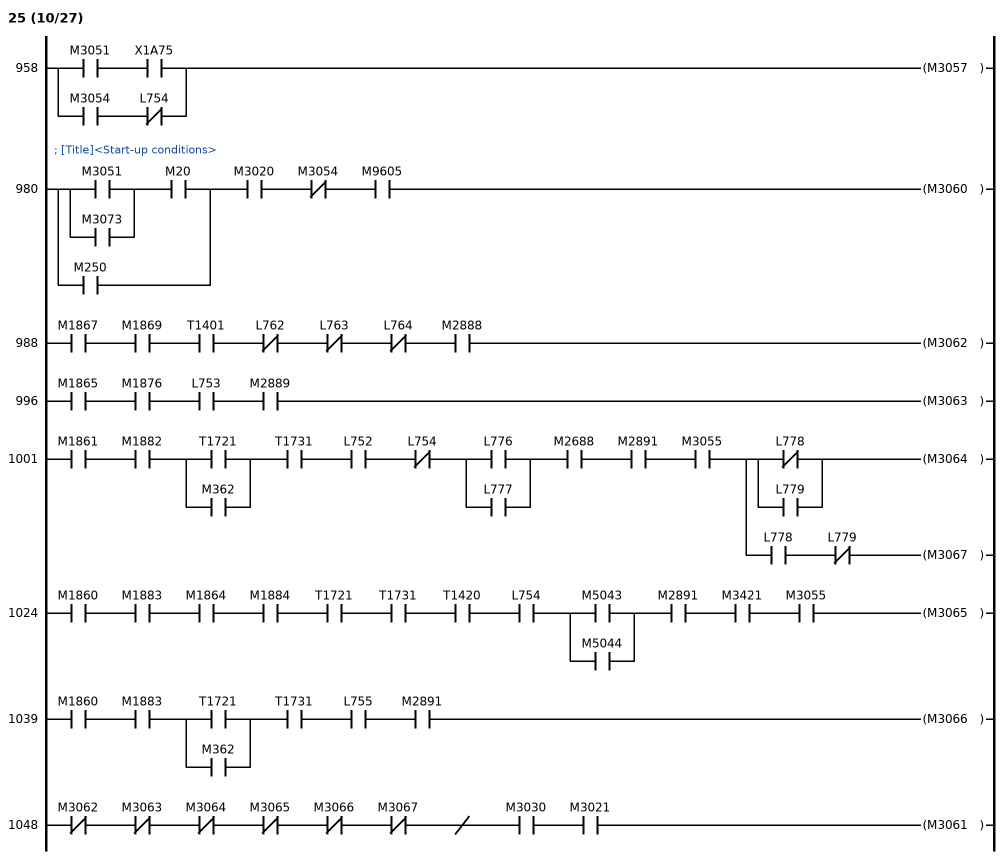
958   LD      M3051
      AND     X1A75
      LD      M3054
      ANI     L754
      ORB
      OUT     M3057
; [Title]<Start-up conditions>
980   LD      M3051
      OR      M3073
      AND     M20
      OR      M250
      AND     M3020
      ANI     M3054
      AND     M9605
      OUT     M3060
988   LD      M1867
      AND     M1869
      AND     T1401
      ANI     L762
      ANI     L763
      ANI     L764
      AND     M2888
      OUT     M3062
996   LD      M1865
      AND     M1876
      AND     L753
      AND     M2889
      OUT     M3063
1001  LD      M1861
      AND     M1882
      LD      T1721
      OR      M362
      ANB
      AND     T1731
      AND     L752
      ANI     L754
      LD      L776
      OR      L777
      ANB
      AND     M2688
      AND     M2891
      AND     M3055
      MPS
      LDI     L778
      OR      L779
      ANB
      OUT     M3064
      MPP
      AND     L778
      ANI     L779
      OUT     M3067
1024  LD      M1860
      AND     M1883
      AND     M1864
      AND     M1884
      AND     T1721
      AND     T1731
      AND     T1420
      AND     L754
      LD      M5043
      OR      M5044
      ANB
      AND     M2891
      AND     M3421
      AND     M3055
      OUT     M3065
1039  LD      M1860
      AND     M1883
      LD      T1721
      OR      M362
      ANB
      AND     T1731
      AND     L755
      AND     M2891
      OUT     M3066
1048  LDI     M3062
      ANI     M3063
      ANI     M3064
      ANI     M3065
      ANI     M3066
      ANI     M3067
      INV
      AND     M3030
      AND     M3021
      OUT     M3061
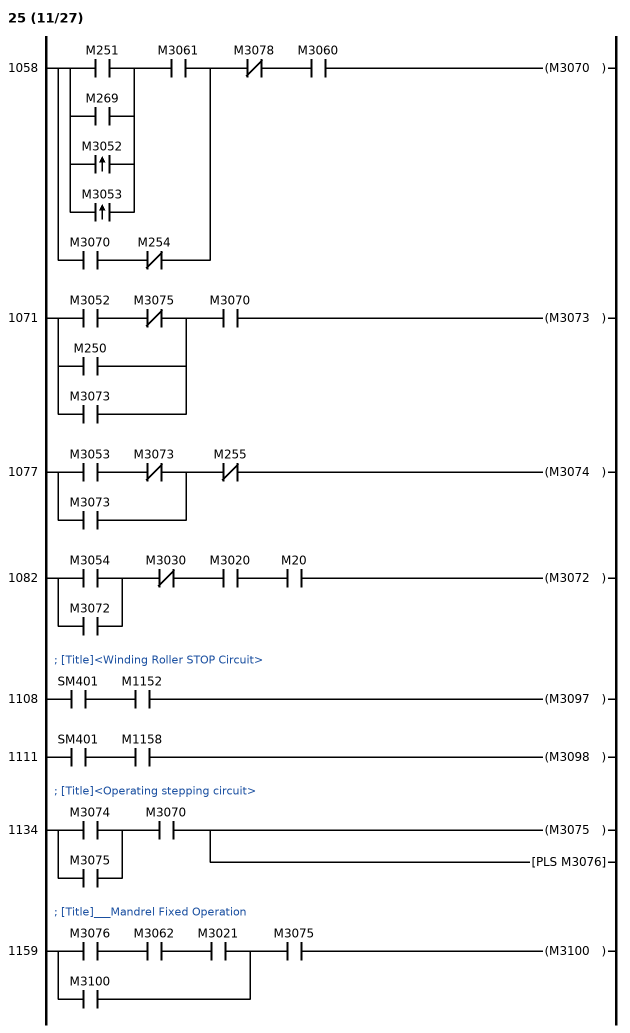
1058  LD      M251
      OR      M269
      ORP     M3052
      ORP     M3053
      AND     M3061
      LD      M3070
      ANI     M254
      ORB
      ANI     M3078
      AND     M3060
      OUT     M3070
1071  LD      M3052
      ANI     M3075
      OR      M250
      OR      M3073
      AND     M3070
      OUT     M3073
1077  LD      M3053
      ANI     M3073
      OR      M3073
      ANI     M255
      OUT     M3074
1082  LD      M3054
      OR      M3072
      ANI     M3030
      AND     M3020
      AND     M20
      OUT     M3072
; [Title]<Winding Roller STOP Circuit>
1108  LD      SM401
      AND     M1152
      OUT     M3097
1111  LD      SM401
      AND     M1158
      OUT     M3098
; [Title]<Operating stepping circuit>
1134  LD      M3074
      OR      M3075
      AND     M3070
      OUT     M3075
      PLS     M3076
; [Title]___Mandrel Fixed Operation
1159  LD      M3076
      AND     M3062
      AND     M3021
      OR      M3100
      AND     M3075
      OUT     M3100
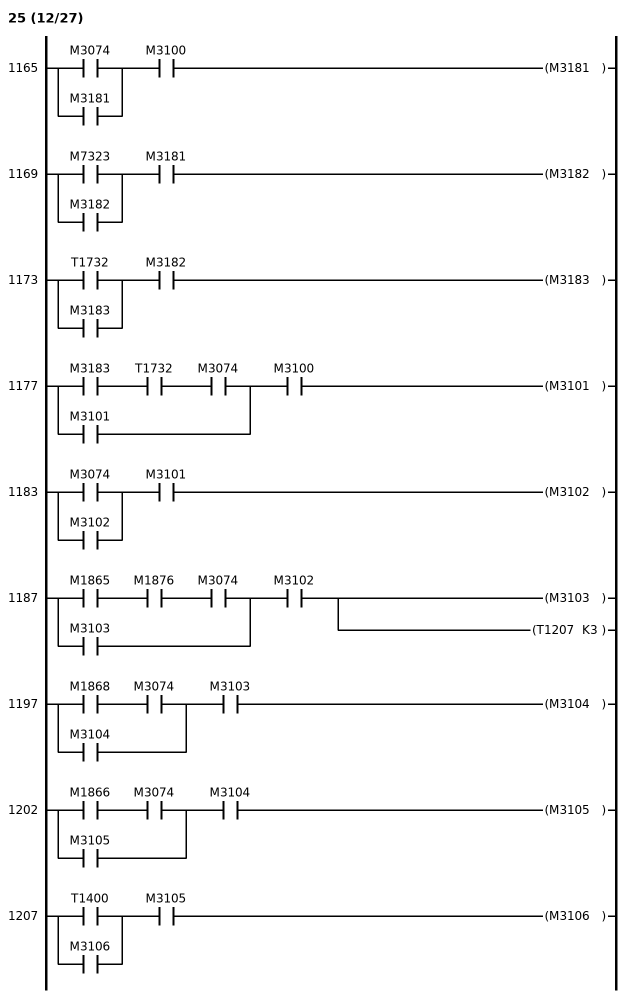
1165  LD      M3074
      OR      M3181
      AND     M3100
      OUT     M3181
1169  LD      M7323
      OR      M3182
      AND     M3181
      OUT     M3182
1173  LD      T1732
      OR      M3183
      AND     M3182
      OUT     M3183
1177  LD      M3183
      AND     T1732
      AND     M3074
      OR      M3101
      AND     M3100
      OUT     M3101
1183  LD      M3074
      OR      M3102
      AND     M3101
      OUT     M3102
1187  LD      M1865
      AND     M1876
      AND     M3074
      OR      M3103
      AND     M3102
      OUT     M3103
      OUT     T1207 K3
1197  LD      M1868
      AND     M3074
      OR      M3104
      AND     M3103
      OUT     M3104
1202  LD      M1866
      AND     M3074
      OR      M3105
      AND     M3104
      OUT     M3105
1207  LD      T1400
      OR      M3106
      AND     M3105
      OUT     M3106
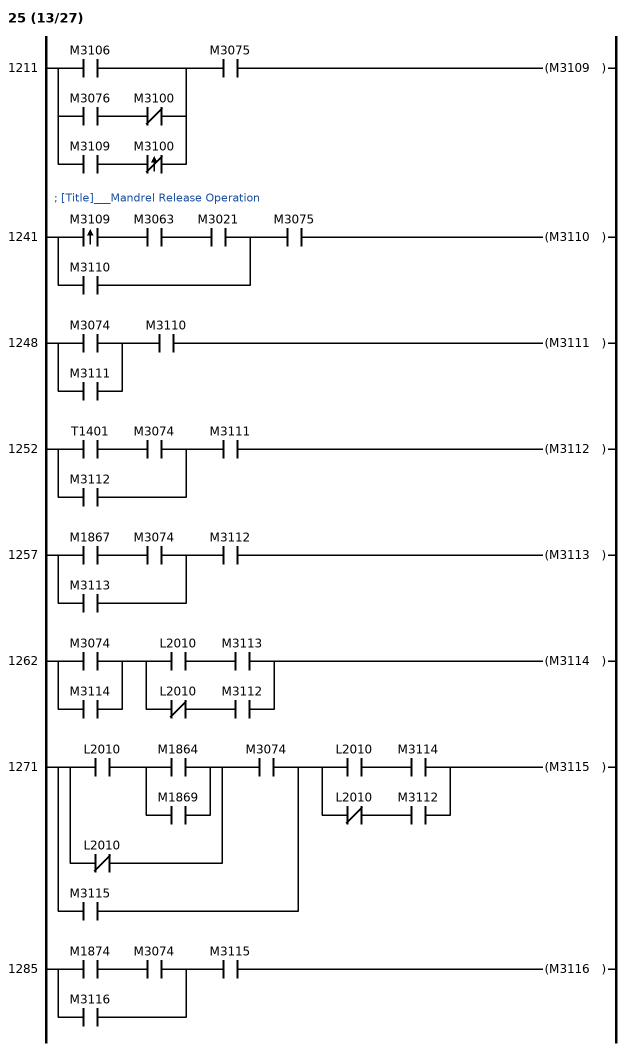
1211  LD      M3106
      LD      M3076
      ANI     M3100
      ORB
      LD      M3109
      ANDPI   M3100
      ORB
      AND     M3075
      OUT     M3109
; [Title]___Mandrel Release Operation
1241  LDP     M3109
      AND     M3063
      AND     M3021
      OR      M3110
      AND     M3075
      OUT     M3110
1248  LD      M3074
      OR      M3111
      AND     M3110
      OUT     M3111
1252  LD      T1401
      AND     M3074
      OR      M3112
      AND     M3111
      OUT     M3112
1257  LD      M1867
      AND     M3074
      OR      M3113
      AND     M3112
      OUT     M3113
1262  LD      M3074
      OR      M3114
      LD      L2010
      AND     M3113
      LDI     L2010
      AND     M3112
      ORB
      ANB
      OUT     M3114
1271  LD      L2010
      LD      M1864
      OR      M1869
      ANB
      ORI     L2010
      AND     M3074
      OR      M3115
      LD      L2010
      AND     M3114
      LDI     L2010
      AND     M3112
      ORB
      ANB
      OUT     M3115
1285  LD      M1874
      AND     M3074
      OR      M3116
      AND     M3115
      OUT     M3116
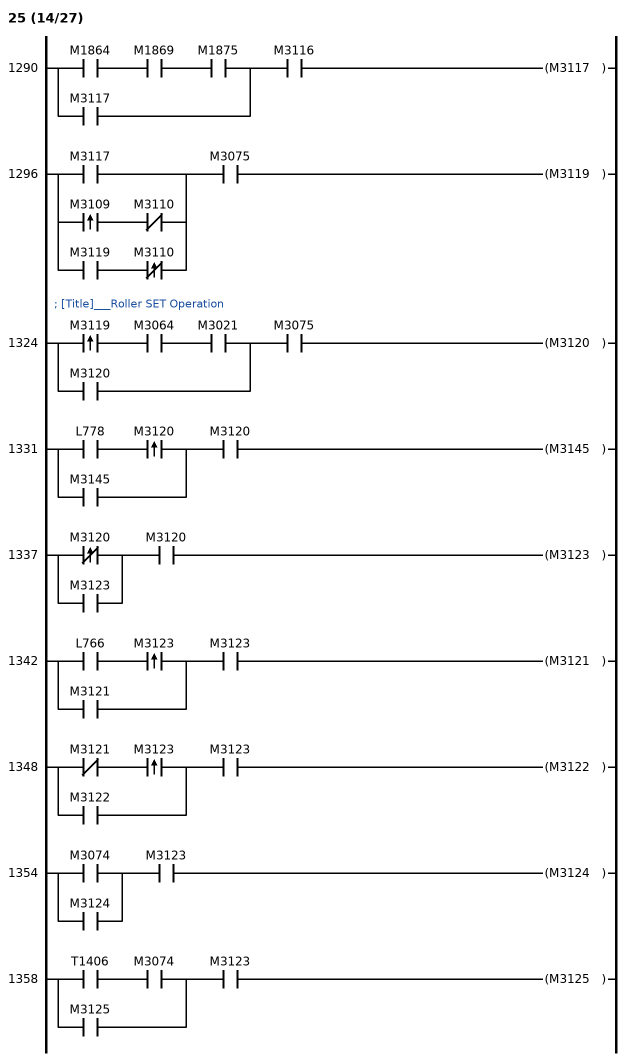
1290  LD      M1864
      AND     M1869
      AND     M1875
      OR      M3117
      AND     M3116
      OUT     M3117
1296  LD      M3117
      LDP     M3109
      ANI     M3110
      ORB
      LD      M3119
      ANDPI   M3110
      ORB
      AND     M3075
      OUT     M3119
; [Title]___Roller SET Operation
1324  LDP     M3119
      AND     M3064
      AND     M3021
      OR      M3120
      AND     M3075
      OUT     M3120
1331  LD      L778
      ANDP    M3120
      OR      M3145
      AND     M3120
      OUT     M3145
1337  LDPI    M3120
      OR      M3123
      AND     M3120
      OUT     M3123
1342  LD      L766
      ANDP    M3123
      OR      M3121
      AND     M3123
      OUT     M3121
1348  LDI     M3121
      ANDP    M3123
      OR      M3122
      AND     M3123
      OUT     M3122
1354  LD      M3074
      OR      M3124
      AND     M3123
      OUT     M3124
1358  LD      T1406
      AND     M3074
      OR      M3125
      AND     M3123
      OUT     M3125
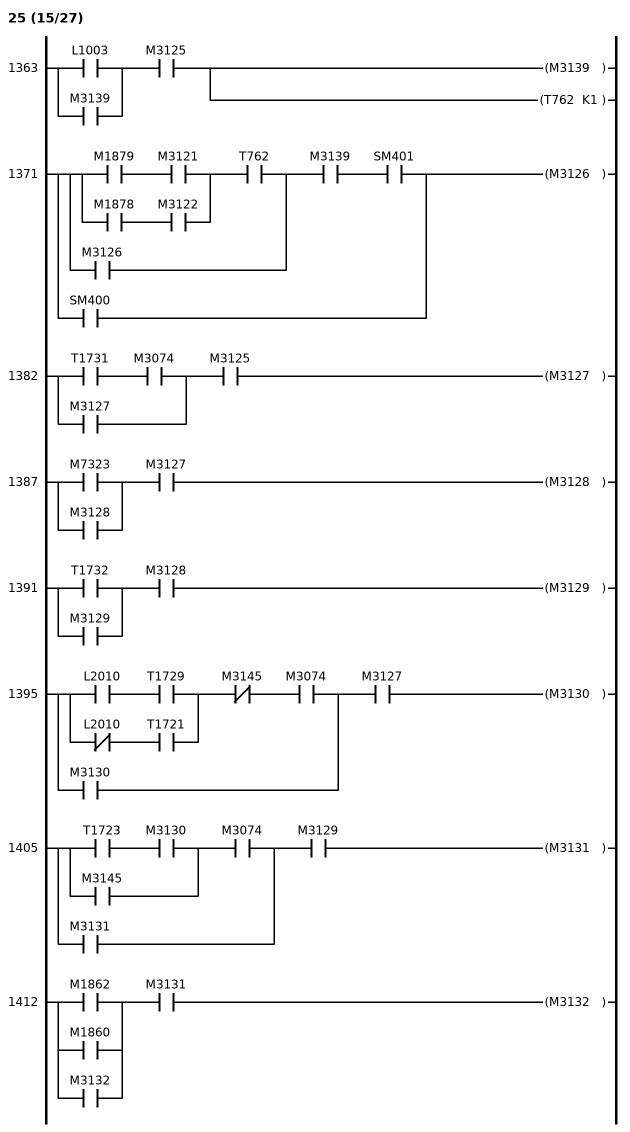
1363  LD      L1003
      OR      M3139
      AND     M3125
      OUT     M3139
      OUT     T762 K1
1371  LD      M1879
      AND     M3121
      LD      M1878
      AND     M3122
      ORB
      AND     T762
      OR      M3126
      AND     M3139
      AND     SM401
      OR      SM400
      OUT     M3126
1382  LD      T1731
      AND     M3074
      OR      M3127
      AND     M3125
      OUT     M3127
1387  LD      M7323
      OR      M3128
      AND     M3127
      OUT     M3128
1391  LD      T1732
      OR      M3129
      AND     M3128
      OUT     M3129
1395  LD      L2010
      AND     T1729
      LDI     L2010
      AND     T1721
      ORB
      ANI     M3145
      AND     M3074
      OR      M3130
      AND     M3127
      OUT     M3130
1405  LD      T1723
      AND     M3130
      OR      M3145
      AND     M3074
      OR      M3131
      AND     M3129
      OUT     M3131
1412  LD      M1862
      OR      M1860
      OR      M3132
      AND     M3131
      OUT     M3132
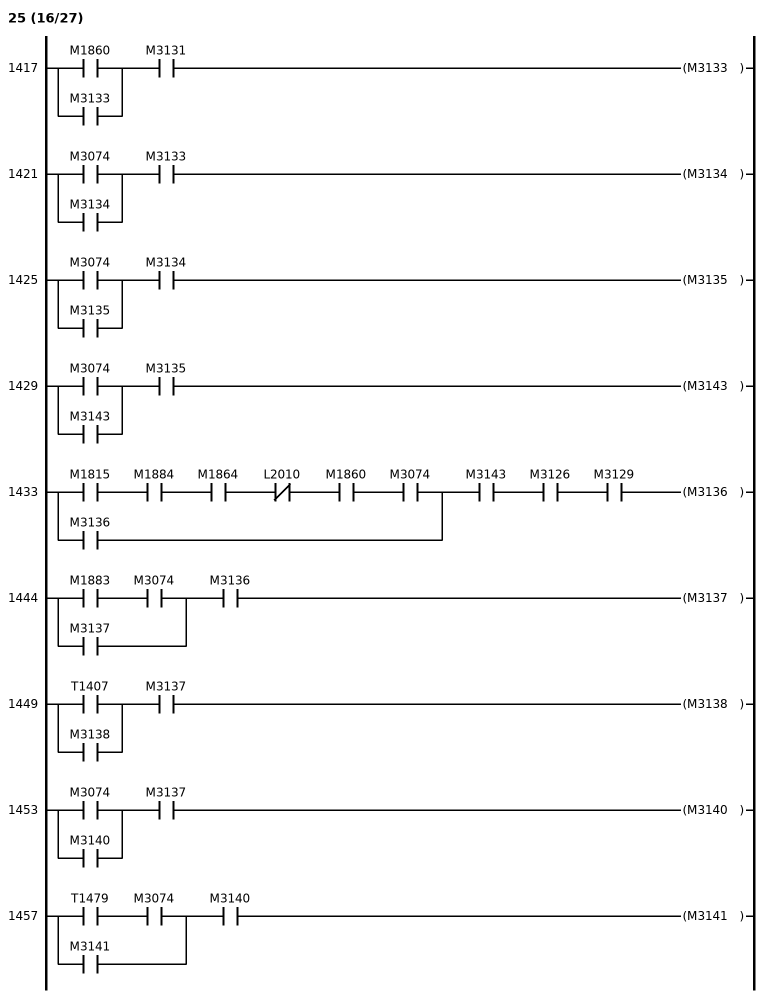
1417  LD      M1860
      OR      M3133
      AND     M3131
      OUT     M3133
1421  LD      M3074
      OR      M3134
      AND     M3133
      OUT     M3134
1425  LD      M3074
      OR      M3135
      AND     M3134
      OUT     M3135
1429  LD      M3074
      OR      M3143
      AND     M3135
      OUT     M3143
1433  LD      M1815
      AND     M1884
      AND     M1864
      ANI     L2010
      AND     M1860
      AND     M3074
      OR      M3136
      AND     M3143
      AND     M3126
      AND     M3129
      OUT     M3136
1444  LD      M1883
      AND     M3074
      OR      M3137
      AND     M3136
      OUT     M3137
1449  LD      T1407
      OR      M3138
      AND     M3137
      OUT     M3138
1453  LD      M3074
      OR      M3140
      AND     M3137
      OUT     M3140
1457  LD      T1479
      AND     M3074
      OR      M3141
      AND     M3140
      OUT     M3141
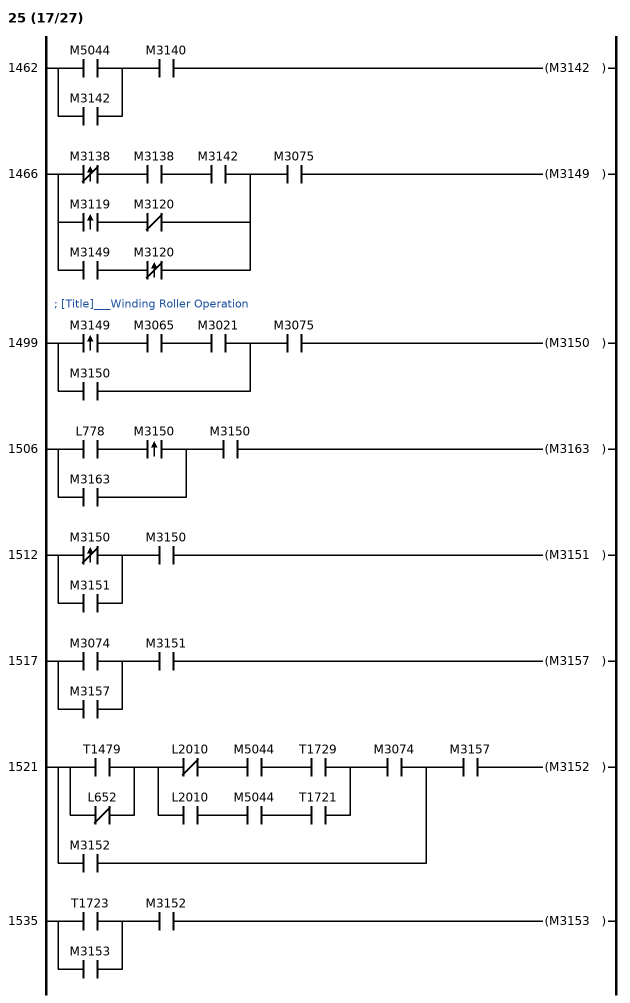
1462  LD      M5044
      OR      M3142
      AND     M3140
      OUT     M3142
1466  LDPI    M3138
      AND     M3138
      AND     M3142
      LDP     M3119
      ANI     M3120
      ORB
      LD      M3149
      ANDPI   M3120
      ORB
      AND     M3075
      OUT     M3149
; [Title]___Winding Roller Operation
1499  LDP     M3149
      AND     M3065
      AND     M3021
      OR      M3150
      AND     M3075
      OUT     M3150
1506  LD      L778
      ANDP    M3150
      OR      M3163
      AND     M3150
      OUT     M3163
1512  LDPI    M3150
      OR      M3151
      AND     M3150
      OUT     M3151
1517  LD      M3074
      OR      M3157
      AND     M3151
      OUT     M3157
1521  LD      T1479
      ORI     L652
      LDI     L2010
      AND     M5044
      AND     T1729
      LD      L2010
      AND     M5044
      AND     T1721
      ORB
      ANB
      AND     M3074
      OR      M3152
      AND     M3157
      OUT     M3152
1535  LD      T1723
      OR      M3153
      AND     M3152
      OUT     M3153
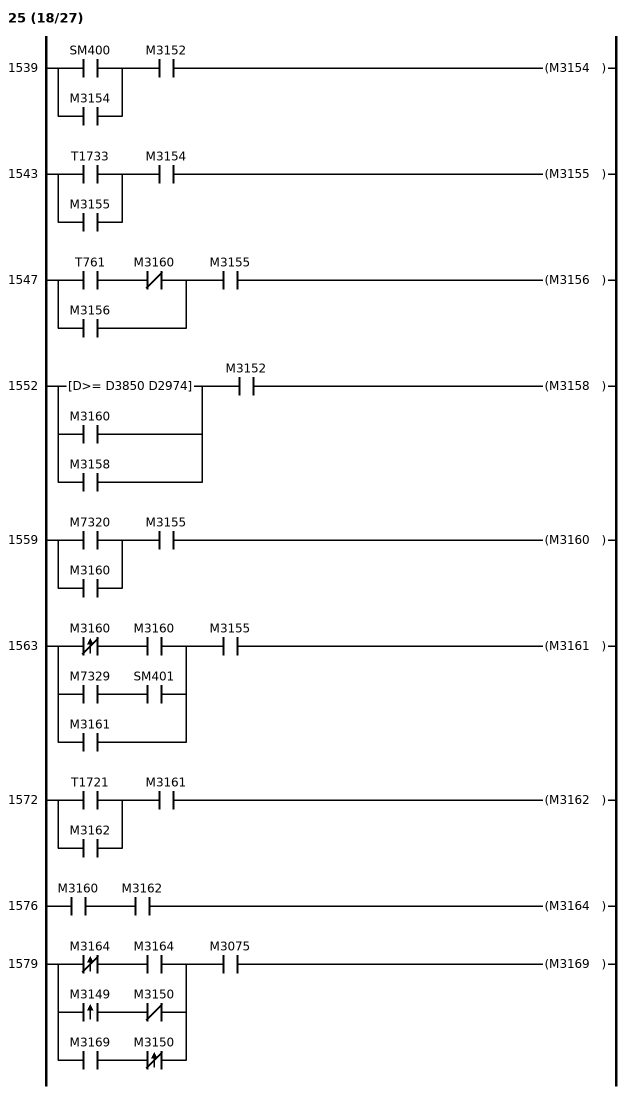
1539  LD      SM400
      OR      M3154
      AND     M3152
      OUT     M3154
1543  LD      T1733
      OR      M3155
      AND     M3154
      OUT     M3155
1547  LD      T761
      ANI     M3160
      OR      M3156
      AND     M3155
      OUT     M3156
1552  LDD>=   D3850 D2974
      OR      M3160
      OR      M3158
      AND     M3152
      OUT     M3158
1559  LD      M7320
      OR      M3160
      AND     M3155
      OUT     M3160
1563  LDPI    M3160
      AND     M3160
      LD      M7329
      AND     SM401
      ORB
      OR      M3161
      AND     M3155
      OUT     M3161
1572  LD      T1721
      OR      M3162
      AND     M3161
      OUT     M3162
1576  LD      M3160
      AND     M3162
      OUT     M3164
1579  LDPI    M3164
      AND     M3164
      LDP     M3149
      ANI     M3150
      ORB
      LD      M3169
      ANDPI   M3150
      ORB
      AND     M3075
      OUT     M3169
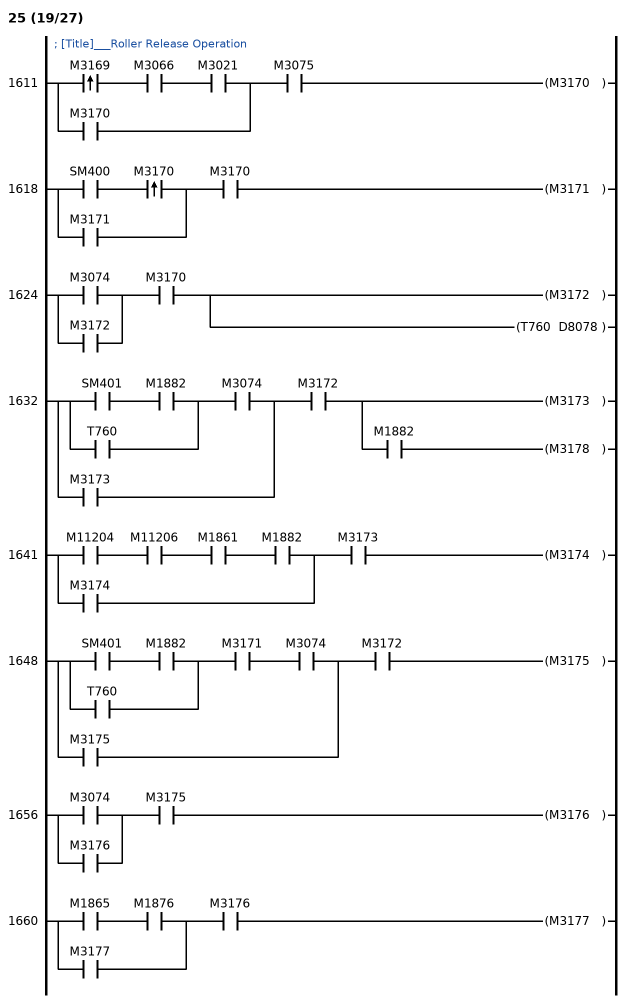
; [Title]___Roller Release Operation
1611  LDP     M3169
      AND     M3066
      AND     M3021
      OR      M3170
      AND     M3075
      OUT     M3170
1618  LD      SM400
      ANDP    M3170
      OR      M3171
      AND     M3170
      OUT     M3171
1624  LD      M3074
      OR      M3172
      AND     M3170
      OUT     M3172
      OUT     T760 D8078
1632  LD      SM401
      AND     M1882
      OR      T760
      AND     M3074
      OR      M3173
      AND     M3172
      OUT     M3173
      AND     M1882
      OUT     M3178
1641  LD      M11204
      AND     M11206
      AND     M1861
      AND     M1882
      OR      M3174
      AND     M3173
      OUT     M3174
1648  LD      SM401
      AND     M1882
      OR      T760
      AND     M3171
      AND     M3074
      OR      M3175
      AND     M3172
      OUT     M3175
1656  LD      M3074
      OR      M3176
      AND     M3175
      OUT     M3176
1660  LD      M1865
      AND     M1876
      OR      M3177
      AND     M3176
      OUT     M3177
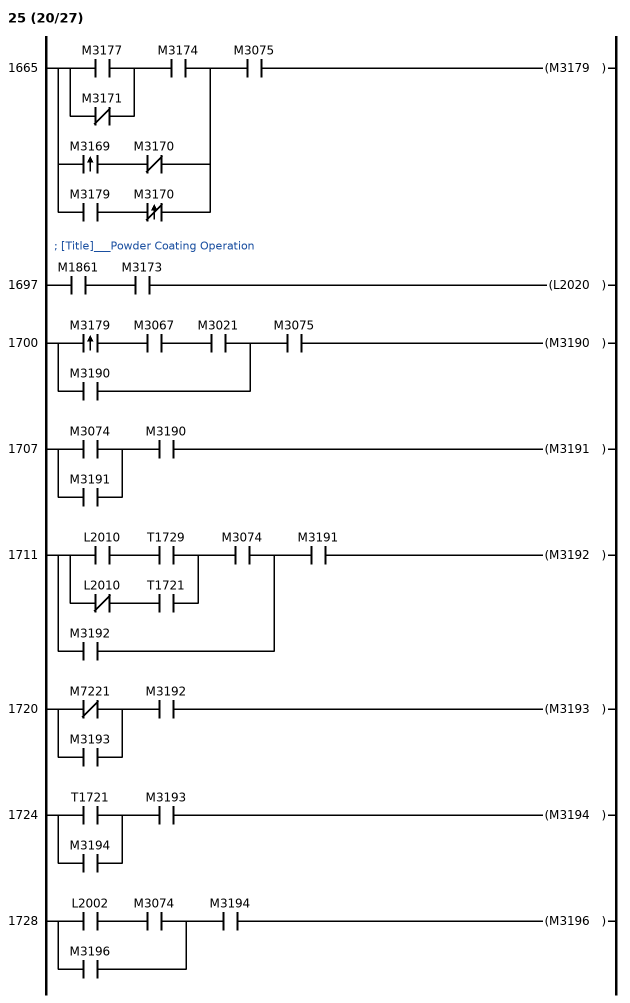
1665  LD      M3177
      ORI     M3171
      AND     M3174
      LDP     M3169
      ANI     M3170
      ORB
      LD      M3179
      ANDPI   M3170
      ORB
      AND     M3075
      OUT     M3179
; [Title]___Powder Coating Operation
1697  LD      M1861
      AND     M3173
      OUT     L2020
1700  LDP     M3179
      AND     M3067
      AND     M3021
      OR      M3190
      AND     M3075
      OUT     M3190
1707  LD      M3074
      OR      M3191
      AND     M3190
      OUT     M3191
1711  LD      L2010
      AND     T1729
      LDI     L2010
      AND     T1721
      ORB
      AND     M3074
      OR      M3192
      AND     M3191
      OUT     M3192
1720  LDI     M7221
      OR      M3193
      AND     M3192
      OUT     M3193
1724  LD      T1721
      OR      M3194
      AND     M3193
      OUT     M3194
1728  LD      L2002
      AND     M3074
      OR      M3196
      AND     M3194
      OUT     M3196
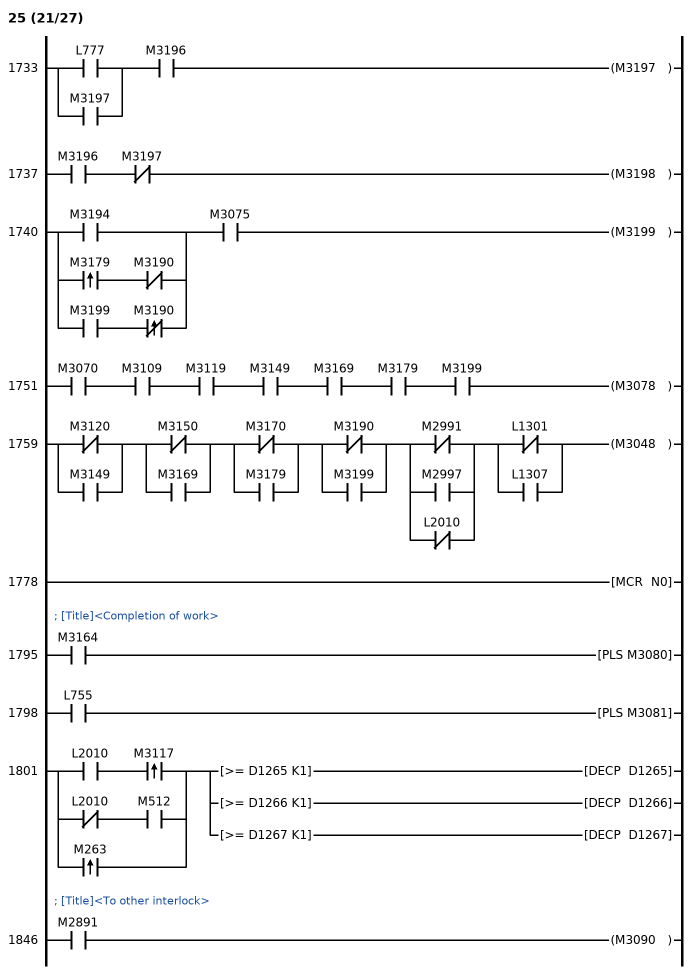
1733  LD      L777
      OR      M3197
      AND     M3196
      OUT     M3197
1737  LD      M3196
      ANI     M3197
      OUT     M3198
1740  LD      M3194
      LDP     M3179
      ANI     M3190
      ORB
      LD      M3199
      ANDPI   M3190
      ORB
      AND     M3075
      OUT     M3199
1751  LD      M3070
      AND     M3109
      AND     M3119
      AND     M3149
      AND     M3169
      AND     M3179
      AND     M3199
      OUT     M3078
1759  LDI     M3120
      OR      M3149
      LDI     M3150
      OR      M3169
      ANB
      LDI     M3170
      OR      M3179
      ANB
      LDI     M3190
      OR      M3199
      ANB
      LDI     M2991
      OR      M2997
      ORI     L2010
      ANB
      LDI     L1301
      OR      L1307
      ANB
      OUT     M3048
1778  MCR     N0
; [Title]<Completion of work>
1795  LD      M3164
      PLS     M3080
1798  LD      L755
      PLS     M3081
1801  LD      L2010
      ANDP    M3117
      LDI     L2010
      AND     M512
      ORB
      ORP     M263
      MPS
      AND>=   D1265 K1
      DECP    D1265
      MRD
      AND>=   D1266 K1
      DECP    D1266
      MPP
      AND>=   D1267 K1
      DECP    D1267
; [Title]<To other interlock>
1846  LD      M2891
      OUT     M3090
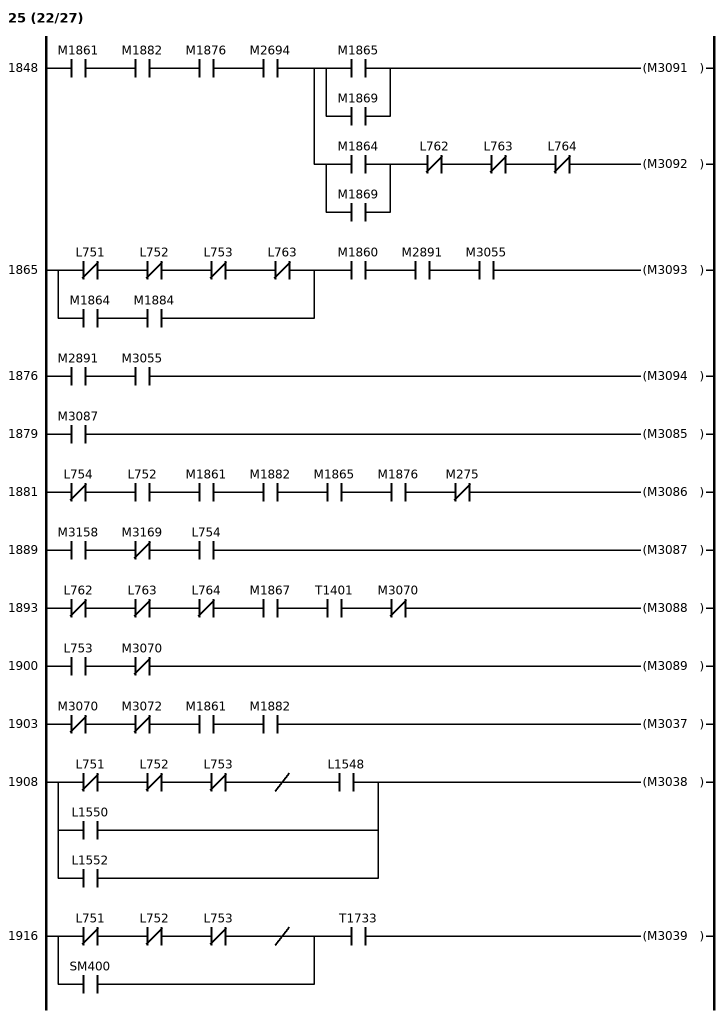
1848  LD      M1861
      AND     M1882
      AND     M1876
      AND     M2694
      MPS
      LD      M1865
      OR      M1869
      ANB
      OUT     M3091
      MPP
      LD      M1864
      OR      M1869
      ANB
      ANI     L762
      ANI     L763
      ANI     L764
      OUT     M3092
1865  LDI     L751
      ANI     L752
      ANI     L753
      ANI     L763
      LD      M1864
      AND     M1884
      ORB
      AND     M1860
      AND     M2891
      AND     M3055
      OUT     M3093
1876  LD      M2891
      AND     M3055
      OUT     M3094
1879  LD      M3087
      OUT     M3085
1881  LDI     L754
      AND     L752
      AND     M1861
      AND     M1882
      AND     M1865
      AND     M1876
      ANI     M275
      OUT     M3086
1889  LD      M3158
      ANI     M3169
      AND     L754
      OUT     M3087
1893  LDI     L762
      ANI     L763
      ANI     L764
      AND     M1867
      AND     T1401
      ANI     M3070
      OUT     M3088
1900  LD      L753
      ANI     M3070
      OUT     M3089
1903  LDI     M3070
      ANI     M3072
      AND     M1861
      AND     M1882
      OUT     M3037
1908  LDI     L751
      ANI     L752
      ANI     L753
      INV
      AND     L1548
      OR      L1550
      OR      L1552
      OUT     M3038
1916  LDI     L751
      ANI     L752
      ANI     L753
      INV
      OR      SM400
      AND     T1733
      OUT     M3039
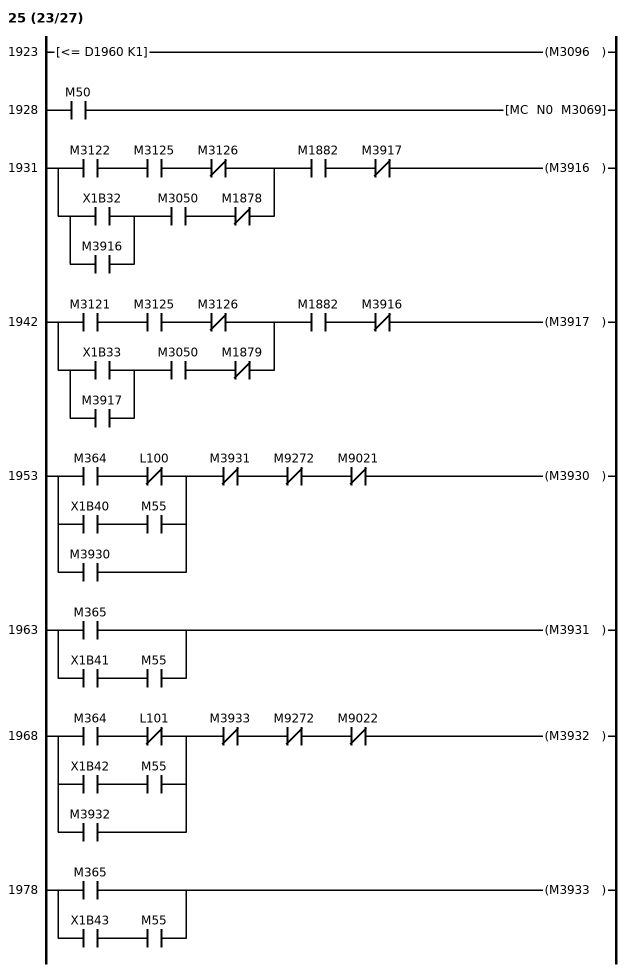
1923  LD<=    D1960 K1
      OUT     M3096
; 
1928  LD      M50
      MC      N0 M3069
1931  LD      M3122
      AND     M3125
      ANI     M3126
      LD      X1B32
      OR      M3916
      AND     M3050
      ANI     M1878
      ORB
      AND     M1882
      ANI     M3917
      OUT     M3916
1942  LD      M3121
      AND     M3125
      ANI     M3126
      LD      X1B33
      OR      M3917
      AND     M3050
      ANI     M1879
      ORB
      AND     M1882
      ANI     M3916
      OUT     M3917
1953  LD      M364
      ANI     L100
      LD      X1B40
      AND     M55
      ORB
      OR      M3930
      ANI     M3931
      ANI     M9272
      ANI     M9021
      OUT     M3930
1963  LD      M365
      LD      X1B41
      AND     M55
      ORB
      OUT     M3931
1968  LD      M364
      ANI     L101
      LD      X1B42
      AND     M55
      ORB
      OR      M3932
      ANI     M3933
      ANI     M9272
      ANI     M9022
      OUT     M3932
1978  LD      M365
      LD      X1B43
      AND     M55
      ORB
      OUT     M3933
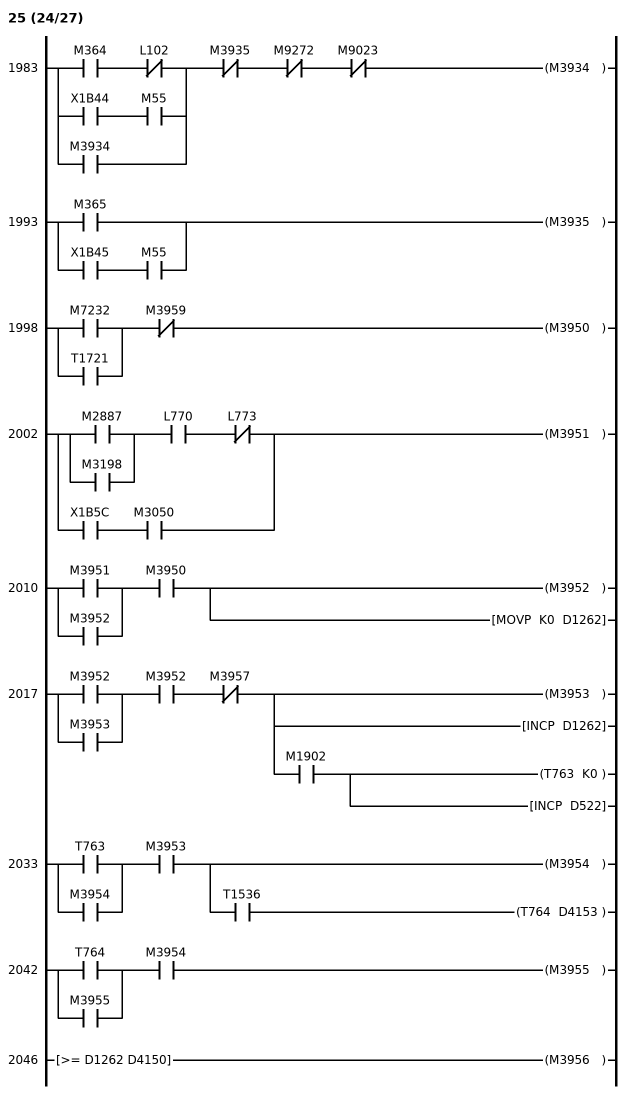
1983  LD      M364
      ANI     L102
      LD      X1B44
      AND     M55
      ORB
      OR      M3934
      ANI     M3935
      ANI     M9272
      ANI     M9023
      OUT     M3934
1993  LD      M365
      LD      X1B45
      AND     M55
      ORB
      OUT     M3935
1998  LD      M7232
      OR      T1721
      ANI     M3959
      OUT     M3950
2002  LD      M2887
      OR      M3198
      AND     L770
      ANI     L773
      LD      X1B5C
      AND     M3050
      ORB
      OUT     M3951
2010  LD      M3951
      OR      M3952
      AND     M3950
      OUT     M3952
      MOVP    K0 D1262
2017  LD      M3952
      OR      M3953
      AND     M3952
      ANI     M3957
      OUT     M3953
      INCP    D1262
      AND     M1902
      OUT     T763 K0
      INCP    D522
2033  LD      T763
      OR      M3954
      AND     M3953
      OUT     M3954
      AND     T1536
      OUT     T764 D4153
2042  LD      T764
      OR      M3955
      AND     M3954
      OUT     M3955
2046  LD>=    D1262 D4150
      OUT     M3956
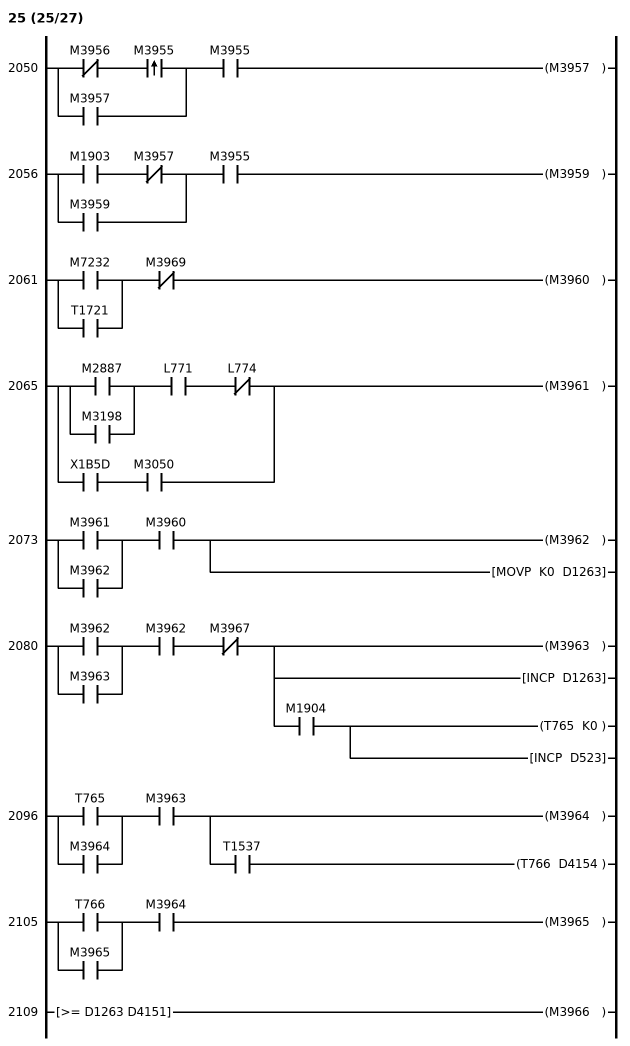
2050  LDI     M3956
      ANDP    M3955
      OR      M3957
      AND     M3955
      OUT     M3957
2056  LD      M1903
      ANI     M3957
      OR      M3959
      AND     M3955
      OUT     M3959
2061  LD      M7232
      OR      T1721
      ANI     M3969
      OUT     M3960
2065  LD      M2887
      OR      M3198
      AND     L771
      ANI     L774
      LD      X1B5D
      AND     M3050
      ORB
      OUT     M3961
2073  LD      M3961
      OR      M3962
      AND     M3960
      OUT     M3962
      MOVP    K0 D1263
2080  LD      M3962
      OR      M3963
      AND     M3962
      ANI     M3967
      OUT     M3963
      INCP    D1263
      AND     M1904
      OUT     T765 K0
      INCP    D523
2096  LD      T765
      OR      M3964
      AND     M3963
      OUT     M3964
      AND     T1537
      OUT     T766 D4154
2105  LD      T766
      OR      M3965
      AND     M3964
      OUT     M3965
2109  LD>=    D1263 D4151
      OUT     M3966
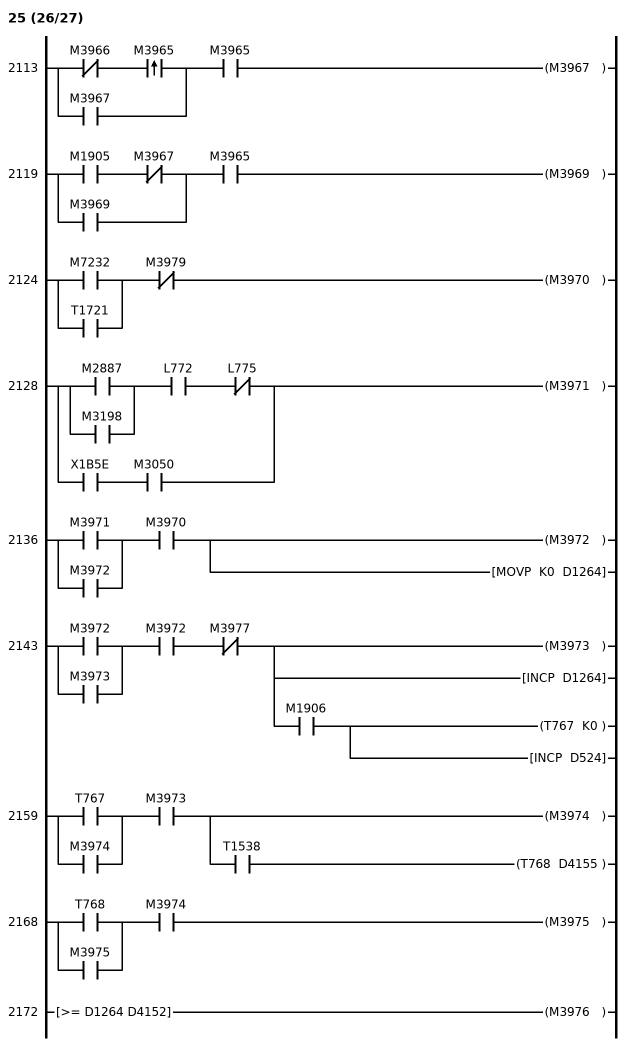
2113  LDI     M3966
      ANDP    M3965
      OR      M3967
      AND     M3965
      OUT     M3967
2119  LD      M1905
      ANI     M3967
      OR      M3969
      AND     M3965
      OUT     M3969
2124  LD      M7232
      OR      T1721
      ANI     M3979
      OUT     M3970
2128  LD      M2887
      OR      M3198
      AND     L772
      ANI     L775
      LD      X1B5E
      AND     M3050
      ORB
      OUT     M3971
2136  LD      M3971
      OR      M3972
      AND     M3970
      OUT     M3972
      MOVP    K0 D1264
2143  LD      M3972
      OR      M3973
      AND     M3972
      ANI     M3977
      OUT     M3973
      INCP    D1264
      AND     M1906
      OUT     T767 K0
      INCP    D524
2159  LD      T767
      OR      M3974
      AND     M3973
      OUT     M3974
      AND     T1538
      OUT     T768 D4155
2168  LD      T768
      OR      M3975
      AND     M3974
      OUT     M3975
2172  LD>=    D1264 D4152
      OUT     M3976
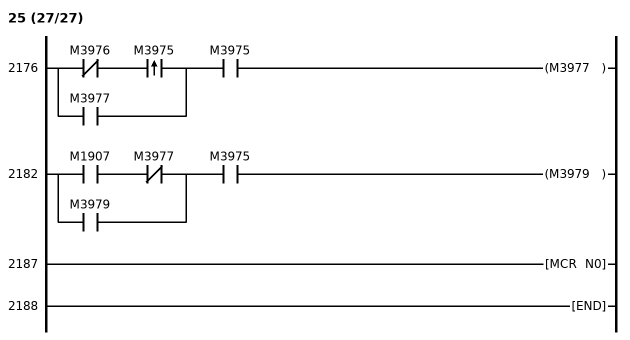
2176  LDI     M3976
      ANDP    M3975
      OR      M3977
      AND     M3975
      OUT     M3977
2182  LD      M1907
      ANI     M3977
      OR      M3979
      AND     M3975
      OUT     M3979
2187  MCR     N0
2188  END
END_PROGRAM

PROGRAM 26
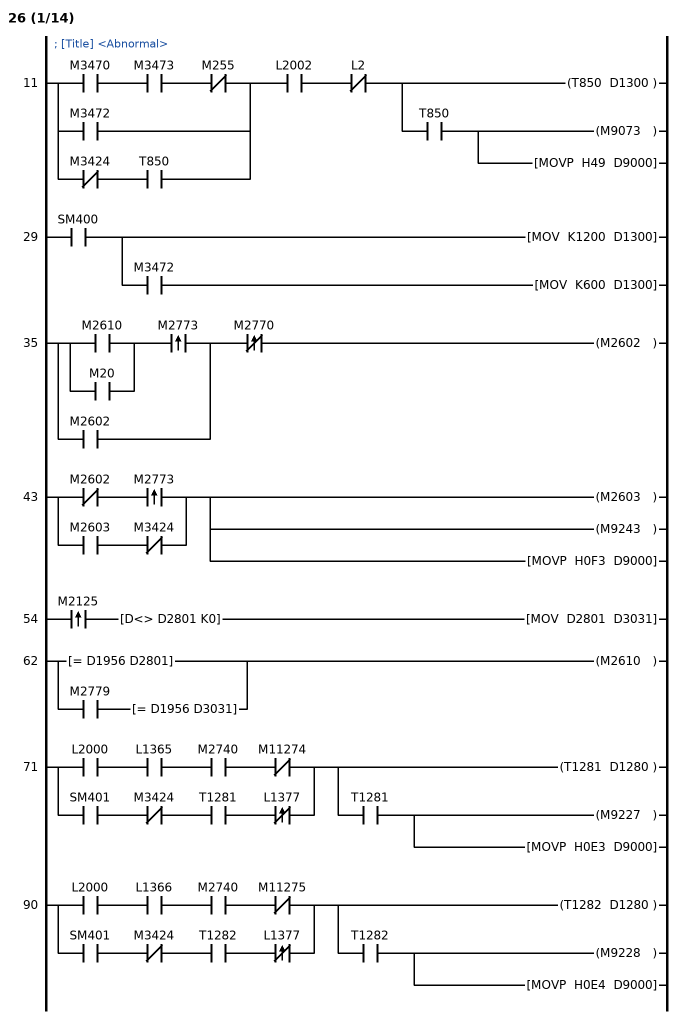
; [Title] <Abnormal>
11    LD      M3470
      AND     M3473
      ANI     M255
      OR      M3472
      LDI     M3424
      AND     T850
      ORB
      AND     L2002
      ANI     L2
      OUT     T850 D1300
      AND     T850
      OUT     M9073
      MOVP    H49 D9000
29    LD      SM400
      MOV     K1200 D1300
      AND     M3472
      MOV     K600 D1300
35    LD      M2610
      OR      M20
      ANDP    M2773
      OR      M2602
      ANDPI   M2770
      OUT     M2602
43    LDI     M2602
      ANDP    M2773
      LD      M2603
      ANI     M3424
      ORB
      OUT     M2603
      OUT     M9243
      MOVP    H0F3 D9000
54    LDP     M2125
      ANDD<>  D2801 K0
      MOV     D2801 D3031
62    LD=     D1956 D2801
      LD      M2779
      AND=    D1956 D3031
      ORB
      OUT     M2610
71    LD      L2000
      AND     L1365
      AND     M2740
      ANI     M11274
      LD      SM401
      ANI     M3424
      AND     T1281
      ANDPI   L1377
      ORB
      OUT     T1281 D1280
      AND     T1281
      OUT     M9227
      MOVP    H0E3 D9000
90    LD      L2000
      AND     L1366
      AND     M2740
      ANI     M11275
      LD      SM401
      ANI     M3424
      AND     T1282
      ANDPI   L1377
      ORB
      OUT     T1282 D1280
      AND     T1282
      OUT     M9228
      MOVP    H0E4 D9000
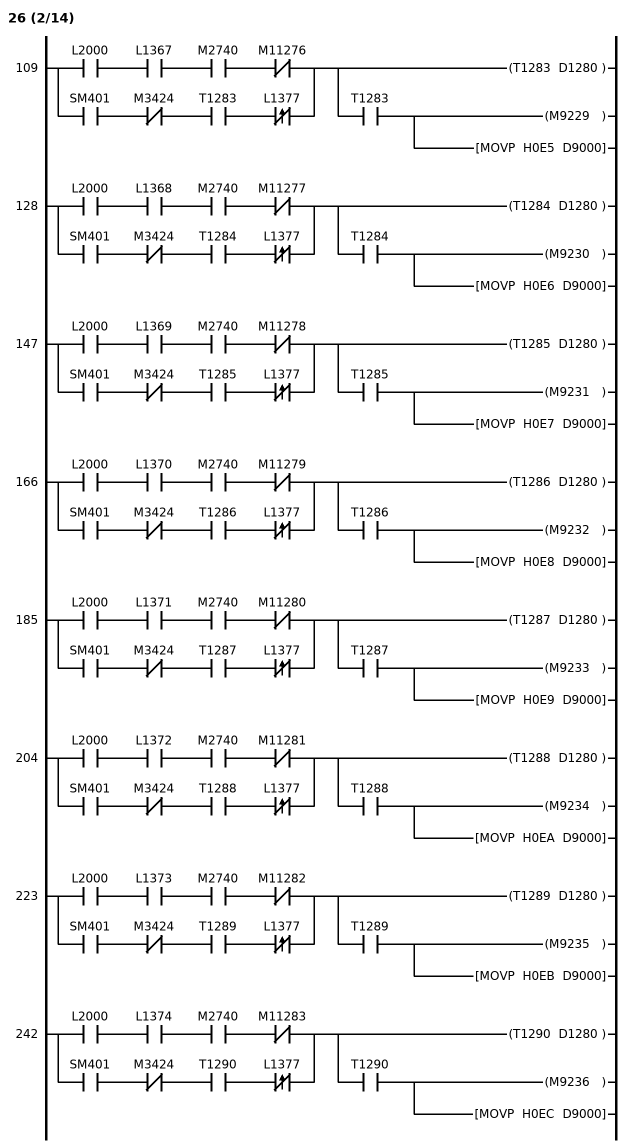
109   LD      L2000
      AND     L1367
      AND     M2740
      ANI     M11276
      LD      SM401
      ANI     M3424
      AND     T1283
      ANDPI   L1377
      ORB
      OUT     T1283 D1280
      AND     T1283
      OUT     M9229
      MOVP    H0E5 D9000
128   LD      L2000
      AND     L1368
      AND     M2740
      ANI     M11277
      LD      SM401
      ANI     M3424
      AND     T1284
      ANDPI   L1377
      ORB
      OUT     T1284 D1280
      AND     T1284
      OUT     M9230
      MOVP    H0E6 D9000
147   LD      L2000
      AND     L1369
      AND     M2740
      ANI     M11278
      LD      SM401
      ANI     M3424
      AND     T1285
      ANDPI   L1377
      ORB
      OUT     T1285 D1280
      AND     T1285
      OUT     M9231
      MOVP    H0E7 D9000
166   LD      L2000
      AND     L1370
      AND     M2740
      ANI     M11279
      LD      SM401
      ANI     M3424
      AND     T1286
      ANDPI   L1377
      ORB
      OUT     T1286 D1280
      AND     T1286
      OUT     M9232
      MOVP    H0E8 D9000
185   LD      L2000
      AND     L1371
      AND     M2740
      ANI     M11280
      LD      SM401
      ANI     M3424
      AND     T1287
      ANDPI   L1377
      ORB
      OUT     T1287 D1280
      AND     T1287
      OUT     M9233
      MOVP    H0E9 D9000
204   LD      L2000
      AND     L1372
      AND     M2740
      ANI     M11281
      LD      SM401
      ANI     M3424
      AND     T1288
      ANDPI   L1377
      ORB
      OUT     T1288 D1280
      AND     T1288
      OUT     M9234
      MOVP    H0EA D9000
223   LD      L2000
      AND     L1373
      AND     M2740
      ANI     M11282
      LD      SM401
      ANI     M3424
      AND     T1289
      ANDPI   L1377
      ORB
      OUT     T1289 D1280
      AND     T1289
      OUT     M9235
      MOVP    H0EB D9000
242   LD      L2000
      AND     L1374
      AND     M2740
      ANI     M11283
      LD      SM401
      ANI     M3424
      AND     T1290
      ANDPI   L1377
      ORB
      OUT     T1290 D1280
      AND     T1290
      OUT     M9236
      MOVP    H0EC D9000
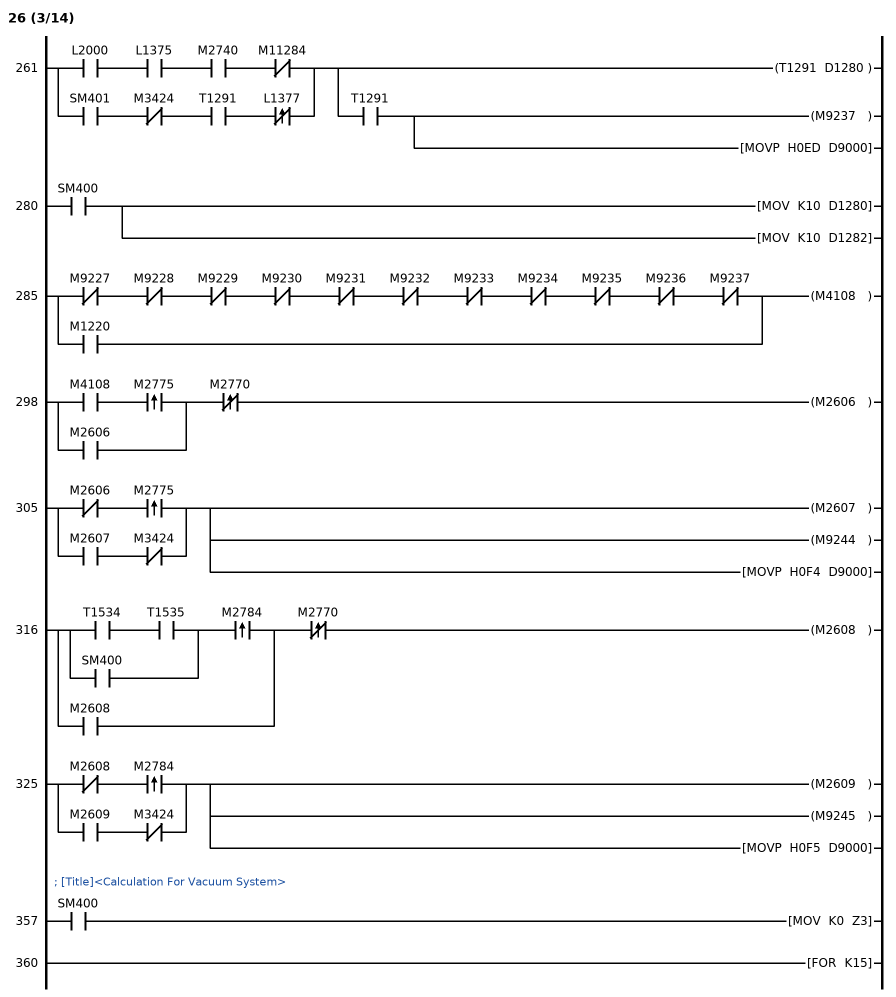
261   LD      L2000
      AND     L1375
      AND     M2740
      ANI     M11284
      LD      SM401
      ANI     M3424
      AND     T1291
      ANDPI   L1377
      ORB
      OUT     T1291 D1280
      AND     T1291
      OUT     M9237
      MOVP    H0ED D9000
280   LD      SM400
      MOV     K10 D1280
      MOV     K10 D1282
285   LDI     M9227
      ANI     M9228
      ANI     M9229
      ANI     M9230
      ANI     M9231
      ANI     M9232
      ANI     M9233
      ANI     M9234
      ANI     M9235
      ANI     M9236
      ANI     M9237
      OR      M1220
      OUT     M4108
298   LD      M4108
      ANDP    M2775
      OR      M2606
      ANDPI   M2770
      OUT     M2606
305   LDI     M2606
      ANDP    M2775
      LD      M2607
      ANI     M3424
      ORB
      OUT     M2607
      OUT     M9244
      MOVP    H0F4 D9000
316   LD      T1534
      AND     T1535
      OR      SM400
      ANDP    M2784
      OR      M2608
      ANDPI   M2770
      OUT     M2608
325   LDI     M2608
      ANDP    M2784
      LD      M2609
      ANI     M3424
      ORB
      OUT     M2609
      OUT     M9245
      MOVP    H0F5 D9000
; [Title]<Calculation For Vacuum System>
357   LD      SM400
      MOV     K0 Z3
360   FOR     K15
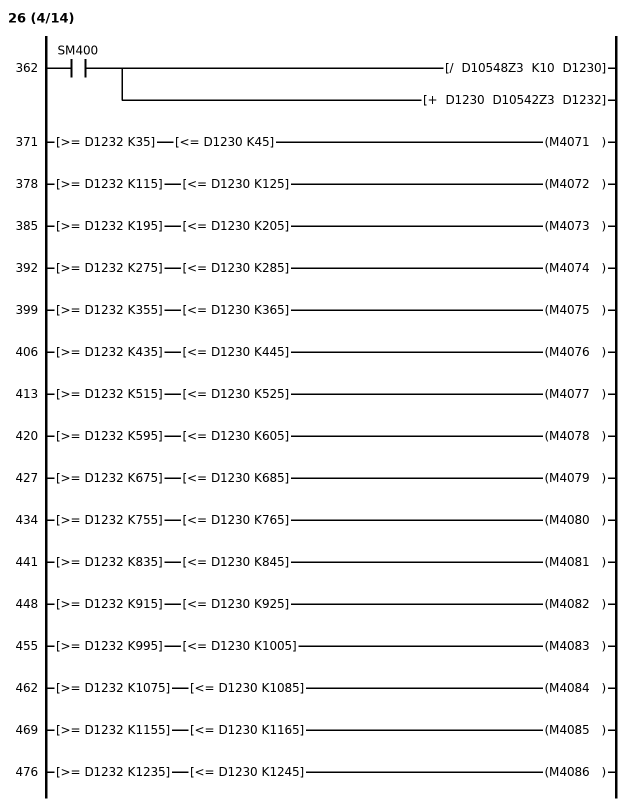
362   LD      SM400
      /       D10548Z3 K10 D1230
      +       D1230 D10542Z3 D1232
371   LD>=    D1232 K35
      AND<=   D1230 K45
      OUT     M4071
378   LD>=    D1232 K115
      AND<=   D1230 K125
      OUT     M4072
385   LD>=    D1232 K195
      AND<=   D1230 K205
      OUT     M4073
392   LD>=    D1232 K275
      AND<=   D1230 K285
      OUT     M4074
399   LD>=    D1232 K355
      AND<=   D1230 K365
      OUT     M4075
406   LD>=    D1232 K435
      AND<=   D1230 K445
      OUT     M4076
413   LD>=    D1232 K515
      AND<=   D1230 K525
      OUT     M4077
420   LD>=    D1232 K595
      AND<=   D1230 K605
      OUT     M4078
427   LD>=    D1232 K675
      AND<=   D1230 K685
      OUT     M4079
434   LD>=    D1232 K755
      AND<=   D1230 K765
      OUT     M4080
441   LD>=    D1232 K835
      AND<=   D1230 K845
      OUT     M4081
448   LD>=    D1232 K915
      AND<=   D1230 K925
      OUT     M4082
455   LD>=    D1232 K995
      AND<=   D1230 K1005
      OUT     M4083
462   LD>=    D1232 K1075
      AND<=   D1230 K1085
      OUT     M4084
469   LD>=    D1232 K1155
      AND<=   D1230 K1165
      OUT     M4085
476   LD>=    D1232 K1235
      AND<=   D1230 K1245
      OUT     M4086
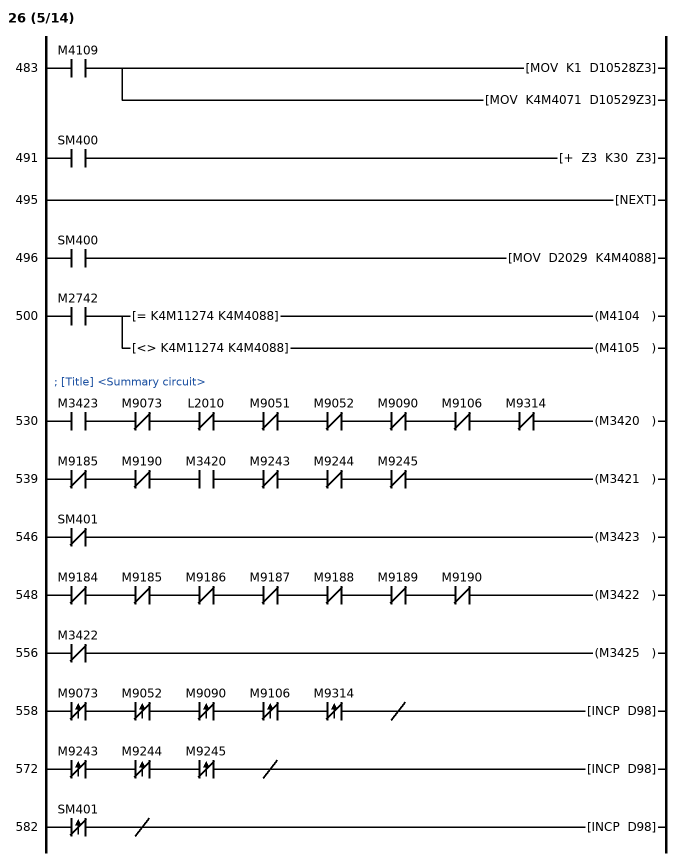
483   LD      M4109
      MOV     K1 D10528Z3
      MOV     K4M4071 D10529Z3
491   LD      SM400
      +       Z3 K30 Z3
495   NEXT
496   LD      SM400
      MOV     D2029 K4M4088
500   LD      M2742
      MPS
      AND=    K4M11274 K4M4088
      OUT     M4104
      MPP
      AND<>   K4M11274 K4M4088
      OUT     M4105
; [Title] <Summary circuit>
530   LD      M3423
      ANI     M9073
      ANI     L2010
      ANI     M9051
      ANI     M9052
      ANI     M9090
      ANI     M9106
      ANI     M9314
      OUT     M3420
539   LDI     M9185
      ANI     M9190
      AND     M3420
      ANI     M9243
      ANI     M9244
      ANI     M9245
      OUT     M3421
546   LDI     SM401
      OUT     M3423
548   LDI     M9184
      ANI     M9185
      ANI     M9186
      ANI     M9187
      ANI     M9188
      ANI     M9189
      ANI     M9190
      OUT     M3422
556   LDI     M3422
      OUT     M3425
558   LDPI    M9073
      ANDPI   M9052
      ANDPI   M9090
      ANDPI   M9106
      ANDPI   M9314
      INV
      INCP    D98
572   LDPI    M9243
      ANDPI   M9244
      ANDPI   M9245
      INV
      INCP    D98
582   LDPI    SM401
      INV
      INCP    D98
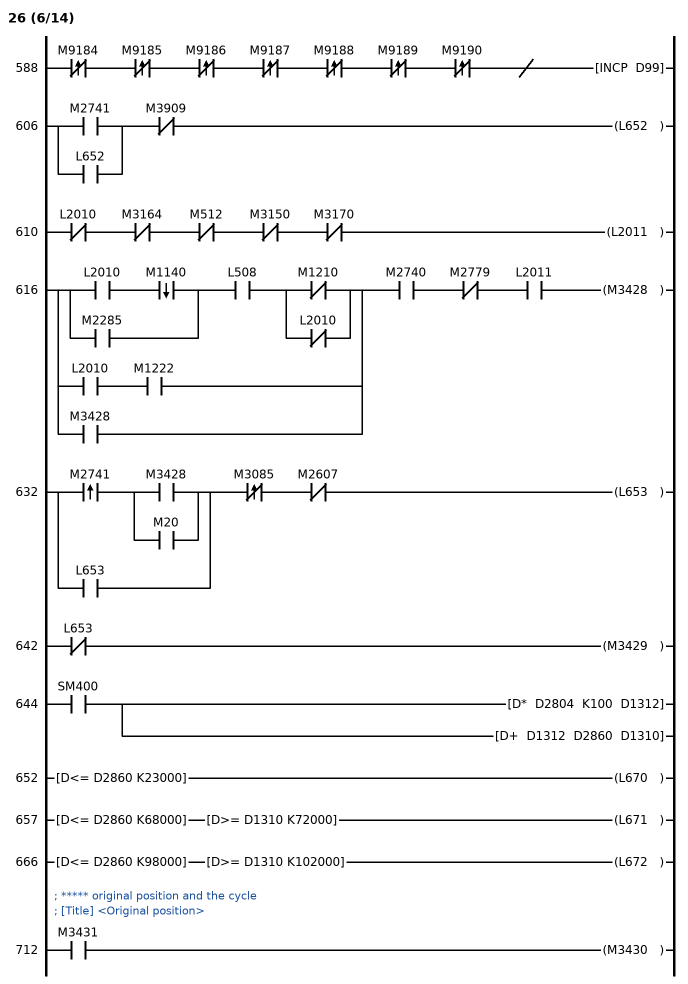
588   LDPI    M9184
      ANDPI   M9185
      ANDPI   M9186
      ANDPI   M9187
      ANDPI   M9188
      ANDPI   M9189
      ANDPI   M9190
      INV
      INCP    D99
606   LD      M2741
      OR      L652
      ANI     M3909
      OUT     L652
610   LDI     L2010
      ANI     M3164
      ANI     M512
      ANI     M3150
      ANI     M3170
      OUT     L2011
616   LD      L2010
      ANDF    M1140
      OR      M2285
      AND     L508
      LDI     M1210
      ORI     L2010
      ANB
      LD      L2010
      AND     M1222
      ORB
      OR      M3428
      AND     M2740
      ANI     M2779
      AND     L2011
      OUT     M3428
632   LDP     M2741
      LD      M3428
      OR      M20
      ANB
      OR      L653
      ANDPI   M3085
      ANI     M2607
      OUT     L653
642   LDI     L653
      OUT     M3429
644   LD      SM400
      D*      D2804 K100 D1312
      D+      D1312 D2860 D1310
652   LDD<=   D2860 K23000
      OUT     L670
657   LDD<=   D2860 K68000
      ANDD>=  D1310 K72000
      OUT     L671
666   LDD<=   D2860 K98000
      ANDD>=  D1310 K102000
      OUT     L672
; ***** original position and the cycle
; [Title] <Original position>
712   LD      M3431
      OUT     M3430
